// TIA Portal V17 export
// export: Created 2025-03-10T13:12:00.5906861Z, ExportSetting WithDefaults, DisplayName Totally Integrated Automation Portal, DisplayVersion V17 Update 8, DisplayName TIA Portal Openness, DisplayVersion V17 Update 8, DisplayName TIA Portal Version Control Interface, DisplayVersion V17, DisplayName SINAMICS Startdrive Advanced, DisplayVersion V17 SP2, DisplayName SINAMICS Startdrive G110M, G120, G120C, G120D, G120P, G115D, DisplayVersion V17 SP2, DisplayName SINAMICS Startdrive G130, G150, S120, S150, SINAMICS MV, S210, DisplayVersion V17 SP2, DisplayName STEP 7 Professional, DisplayVersion V17 Update 8, DisplayName SINUMERIK ONE STEP 7 Toolbox, DisplayVersion V17 Update 12, DisplayName SINUMERIK 840D sl STEP 7 Toolbox, DisplayVersion V17 Update 12, DisplayName STEP 7 Safety, DisplayVersion V17 Update 6, DisplayName WinCC Advanced, DisplayVersion V17 Update 8
TYPE "LBP_typeModularMcpLedAttribute"
TITLE = Modular MCP image / Imagen de MCP modulares / Abbild modulare MCP
// User data type for LBP_typeModularMcpKeypadRecord (sub type) / Tipo de datos de usuario para LBP_typeModularMcpKeypadRecord (subtipo) / Anwenderdatentyp für LBP_typeModularMcpKeypadRecord (Untertyp)
// stored: IsFailsafeCompliant false
   STRUCT
      keyIndex : USInt;   // Tastenindex / index of key / Índice de tecla
      red : USInt;   // Intensität der roten LED / intensity of red LED / Intensidad del LED rojo
      green : USInt;   // Intensität der grünen LED / intensity of green LED / Intensidad del LED verde
      blue : USInt;   // Intensität der blauen LED / intensity of blue LED / Intensidad del LED azul
   END_STRUCT;
END_TYPE
